(* This version of the block is self contained. Minimizes wiring.*)
FUNCTION_BLOCK FB_ExampleDeviceSM_All
VAR_INPUT
	cBase: UDINT;
END_VAR
VAR_OUTPUT
END_VAR
VAR_IN_OUT
	
END_VAR
VAR
	stDevice	:	ST_Device;
	fbGovernor	:	FB_LinearGovernor;
	mcPower	:	MC_Power;
	mcStop: MC_Stop;
	mcAbsolute	:	MC_MoveAbsolute;
	fbBPTM	:	BeamParameterTransitionManager;
	xStartMove: BOOL;
	
	stCheckState: ST_DeviceState;
	stTargetState	:	ST_DeviceState; //Target device state

END_VAR
VAR PERSISTENT
	nLastActiveState	:	UDINT;
END_VAR

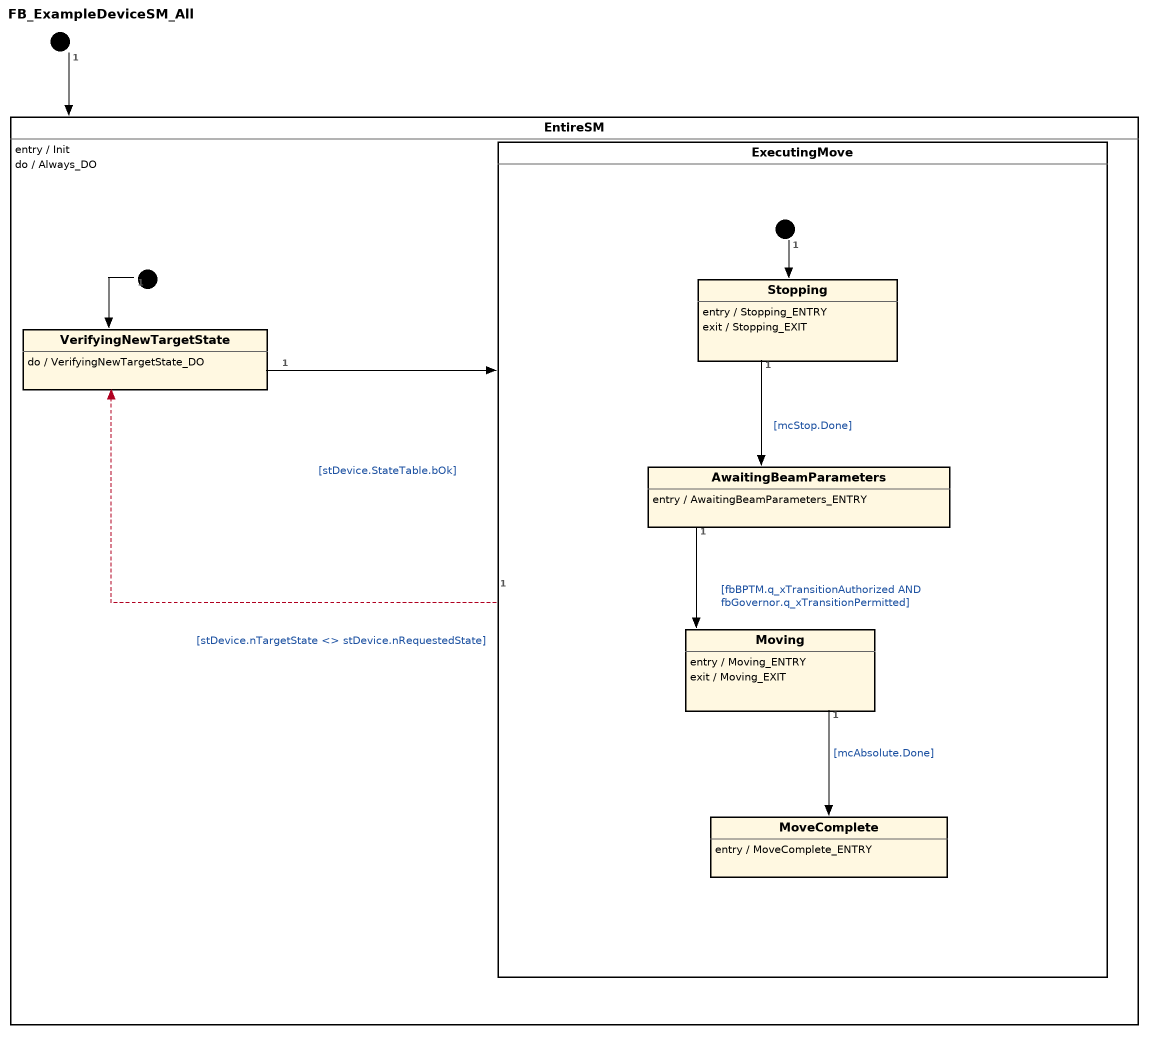
STATECHART FB_ExampleDeviceSM_1  // abortable
    START StartState3
    COMPOSITE STATE EntireSM
        entry / Init
        do / Always_DO
        START StartState1
        COMPOSITE STATE ExecutingMove
            START StartState2
            STATE Stopping
                entry / Stopping_ENTRY
                exit / Stopping_EXIT
            STATE AwaitingBeamParameters
                entry / AwaitingBeamParameters_ENTRY
            STATE Moving
                entry / Moving_ENTRY
                exit / Moving_EXIT
            STATE MoveComplete
                entry / MoveComplete_ENTRY
            StartState2 -> Stopping  // priority 1, on completion
            Stopping -> AwaitingBeamParameters [mcStop.Done] // priority 1, rising edge
            AwaitingBeamParameters -> Moving [fbBPTM.q_xTransitionAuthorized AND fbGovernor.q_xTransitionPermitted] // priority 1, rising edge
            Moving -> MoveComplete [mcAbsolute.Done] // priority 1, rising edge
        END_STATE
        STATE VerifyingNewTargetState
            do / VerifyingNewTargetState_DO
        StartState1 -> VerifyingNewTargetState  // priority 1, on completion
        ExecutingMove -> VerifyingNewTargetState [stDevice.nTargetState <> stDevice.nRequestedState] // priority 1, exception, rising edge
        VerifyingNewTargetState -> ExecutingMove [stDevice.StateTable.bOk] // priority 1
    END_STATE
    StartState3 -> EntireSM  // priority 1, on completion
END_STATECHART

ACTION Always_DO:
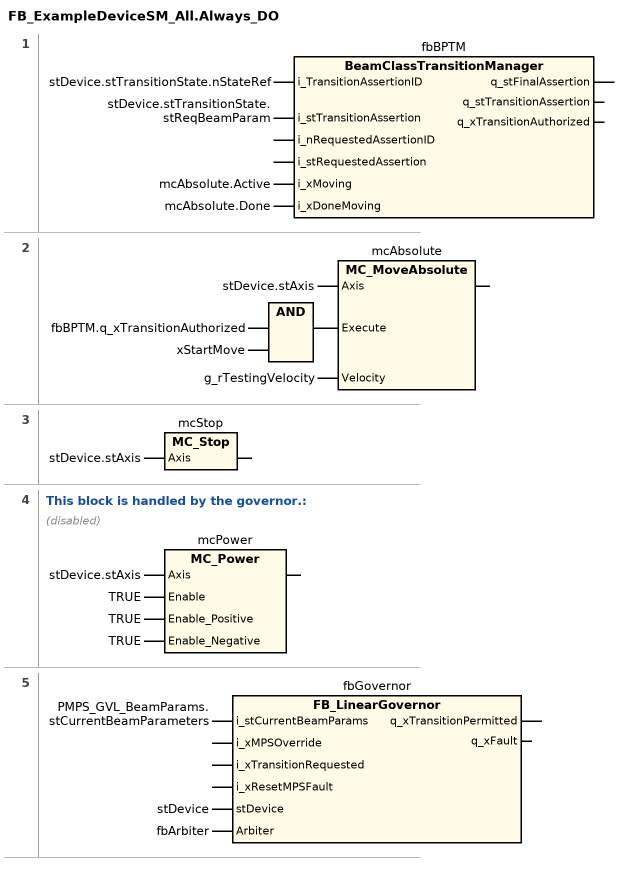
// NETWORK 1
fbBPTM(
    i_TransitionAssertionID := stDevice.stTransitionState.nStateRef,
    i_stTransitionAssertion := stDevice.stTransitionState.stReqBeamParam,
    i_xMoving := mcAbsolute.Active,
    i_xDoneMoving := mcAbsolute.Done); // BeamClassTransitionManager

// NETWORK 2
mcAbsolute(
    Axis := stDevice.stAxis,
    Execute := fbBPTM.q_xTransitionAuthorized AND xStartMove,
    Velocity := g_rTestingVelocity); // MC_MoveAbsolute

// NETWORK 3
mcStop(Axis := stDevice.stAxis); // MC_Stop

// NETWORK 4 (disabled)
// label: This block is handled by the governor.
// mcPower(Axis := stDevice.stAxis, Enable := TRUE, Enable_Positive := TRUE, Enable_Negative := TRUE); // MC_Power

// NETWORK 5
fbGovernor(
    i_stCurrentBeamParams := PMPS_GVL_BeamParams.stCurrentBeamParameters,
    stDevice := stDevice,
    Arbiter := fbArbiter); // FB_LinearGovernor
END_ACTION

ACTION AwaitingBeamParameters_ENTRY:
fbBPTM.i_stRequestedAssertion := stTargetState.stReqBeamParam;
fbBPTM.i_nRequestedAssertionID := stTargetState.nStateRef;

//Tell the governor that we're trying to move.
fbGovernor.i_xTransitionRequested := TRUE;
END_ACTION

ACTION Init:

//Safe State
stDevice.nSafeState := cBase;
stDevice.nTransitionState := cBase+100;

//Initialize the State Table
stDevice.StateTable.A_Reset();

//Device State Table Instantiation
F_SetStateParams(
	nStateRef := stDevice.nSafeState,
	rPosition := 0,
	rTolerance := 10,
	stBeamParams := PMPS_GVL_BeamParams.cstFullBeam,
	Table := stDevice.StateTable
);
F_SetStateParams(
	nStateRef := cBase + 1,
	rPosition := 100,
	rTolerance := 10,
	stBeamParams := F_SetBeamParams(
		fAtt := 20,
		fPP_mJ := 1,
		fLower_eV := 0,
		fUpper_eV := 1500,
		nRate := 10
		),
	Table := stDevice.StateTable
);
F_SetStateParams(
	nStateRef := cBase + 2,
	rPosition := 200,
	rTolerance := 10,
	stBeamParams := F_SetBeamParams(
		fAtt := 30,
		fPP_mJ := 1,
		fLower_eV := 0,
		fUpper_eV := 1500,
		nRate := 10
		),
	Table := stDevice.StateTable
);
F_SetStateParams(
	nStateRef := cBase + 3,
	rPosition := 300,
	rTolerance := 10,
	stBeamParams := F_SetBeamParams(
		fAtt := 20,
		fPP_mJ := 1,
		fLower_eV := 0,
		fUpper_eV := 1500,
		nRate := 10
		),
	Table := stDevice.StateTable
);

F_SetStateParams(
	nStateRef := stDevice.nTransitionState,
	rPosition := 300,
	rTolerance := 10,
	stBeamParams := F_SetBeamParams(
		fAtt := 100,
		fPP_mJ := 0,
		fLower_eV := 0,
		fUpper_eV := 1500,
		nRate := 0
		),
	Table := stDevice.StateTable
);

stDevice.StateTable.A_Lookup(
	key := stDevice.nTransitionState,
	getValue => stDevice.stTransitionState
);

//Need an initialization routine for setting the active state
//Check if the device is at the last known state
//If the device is within the state boundaries, it's considered to be in that state
stDevice.StateTable.A_Lookup(key:= nLastActiveState);
IF stDevice.StateTable.bOk THEN
	stCheckState := stDevice.StateTable.getValue;
ELSE
	stCheckState := stDevice.stTransitionState; //This needs to be safer <TODO>
END_IF

IF stDevice.stAxis.NcToPlc.ActPos <= stCheckstate.rPosition + stCheckState.rTolerance AND
	stDevice.stAxis.NcToPlc.ActPos >= stCheckState.rPosition - stCheckState.rTolerance THEN
	stDevice.nActiveState := nLastActiveState;
ELSE
	stDevice.nActiveState := stDevice.nTransitionState;
END_IF

//Simulation Hardware Limit Switches
stDevice.i_xHiLim := TRUE;
stDevice.i_xLoLim := TRUE;
END_ACTION

ACTION Initialize:

END_ACTION

ACTION MoveComplete_ENTRY:
//Clear transition request
fbGovernor.i_xTransitionRequested := FALSE;
//Latch active state
stDevice.nActiveState := stDevice.nTargetState;
nLastActiveState := stDevice.nActiveState;
END_ACTION

ACTION Moving_ENTRY:
xStartMove := TRUE;
mcAbsolute.Position := stTargetState.rPosition;
END_ACTION

ACTION Moving_EXIT:
xStartMove := FALSE;
END_ACTION

ACTION NewMove_ENTRY:

END_ACTION

ACTION Stopping_ENTRY:
mcStop.Execute := TRUE;
END_ACTION

ACTION Stopping_EXIT:
mcStop.Execute := FALSE;
END_ACTION

ACTION VerifyingNewTargetState_DO:
stDevice.StateTable.A_Lookup(
	key := stDevice.nRequestedState
);

IF stDevice.StateTable.bOk THEN
	stTargetState := stDevice.StateTable.getValue;
	stDevice.nTargetState := stDevice.nRequestedState;
ELSE
	; //log ignored state/ generate an error? <TODO>
END_IF
END_ACTION

END_FUNCTION_BLOCK

(* stored: Version 1.1.0.1, ProductVersion 3.1.4022.12
   POU FB_ExampleDeviceSM_All: Id {77b40f44-00cc-0c50-289c-0c68630377d8}, SpecialFunc None
   Action Always_DO: Id {27e65919-5439-0ac6-21c6-48913d6316f0}
   Action AwaitingBeamParameters_ENTRY: Id {11998768-796a-0ae7-236e-b6d3653f5325}
   Action Init: Id {36a0d24a-22c6-0d0b-1731-1ec66408ff3d}
   Action Initialize: Id {2aa2d54e-87a7-0e29-2ee0-00f6a86237f0}
   Action MoveComplete_ENTRY: Id {6d810ec6-c799-0cbf-2c82-fd4df76e05df}
   Action Moving_ENTRY: Id {309aec0a-c30e-0230-3875-12210036fc1f}
   Action Moving_EXIT: Id {9531dfcf-0b19-0cb7-2f5f-cb82ea7a90dc}
   Action NewMove_ENTRY: Id {d8b0ad57-77e3-0f41-0c64-60320e6d9333}
   Action Stopping_ENTRY: Id {9349f20c-976c-005a-3b7a-9a689850c9c0}
   Action Stopping_EXIT: Id {af8aa562-fd2e-0ca9-251c-e85c3ea25f69}
   Action VerifyingNewTargetState_DO: Id {a05533c0-b048-0735-3044-b56f29dc3283} *)
